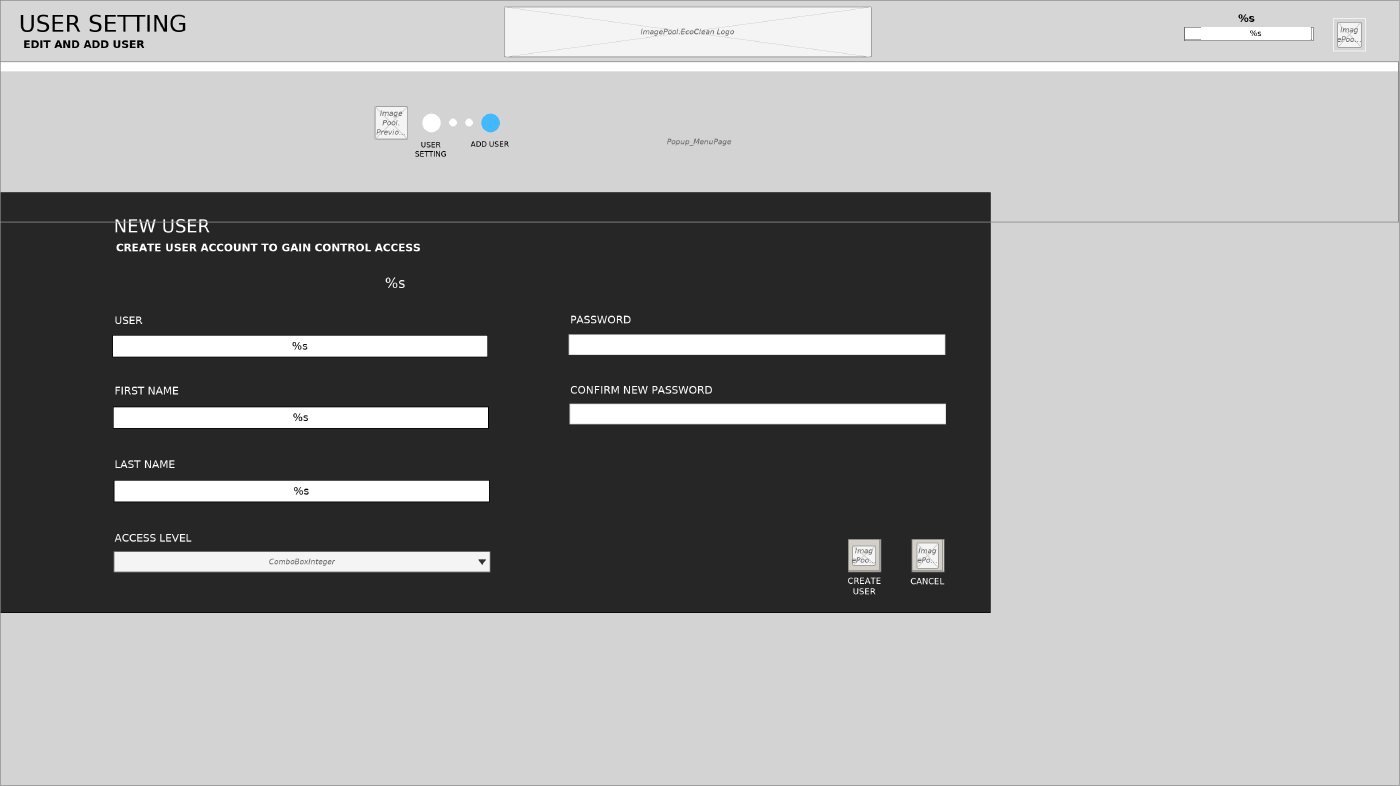
VISUALIZATION AddNewUser_Page  // 1920x1079
    Rectangle (0,98 1920x981)
    Rectangle (0,63 1920x26)
        p3528305787: HMI_Ctrl.ANIMATION3
    Rectangle (0,0 1919x85)
    Label (23,6 310x53), "USER SETTING"
    Label (29,49 320x24), "EDIT AND ADD USER"
    Group (1828,25 45x45)
        OnMouseClick: toggle HMI_Ctrl.MenuButton
        RoundedRectangle (0,0 45x45), colour toggle: HMI_Ctrl.MenuButton
        Image (6,5 33x35), image: ImagePool.Menu Button
    Image (691,9 504x69), image: ImagePool.EcoClean Logo
    Group (1621,14 180x42)
        Rectangle (0,0 177x22), "%s", text variable: DSLocalSystemTimeML.sCurrentDT24Hr_General
        Button (3,23 177x19), image: VisuSymbols.Symbols.AddUser
        Rectangle (26,23 150x18), "%s", text variable: fbHmiTF1800_UserlevelManagement.dsHmiUserStatus_Active.sLoginName
    Rectangle (0,264 1358x577)
    Label (153,284 221x53), "NEW USER"
    Label (156,321 609x38), "CREATE USER ACCOUNT TO GAIN CONTROL ACCESS"
    Label (154,712 216x53), "ACCESS LEVEL"
    ComboBoxInteger (156,757 516x28), variable: sUM_NewUserGroupId, text list: 'TextList_AccessLevel'
    Label (154,611 216x53), "LAST NAME"
    Label (154,409 123x62), "USER"
    Label (154,510 216x53), "FIRST NAME"
    Label (779,408 195x62), "PASSWORD"
    Label (779,509 229x53), "CONFIRM NEW PASSWORD"
    Textfield (781,554 516x28), text variable: sUM_ConfirmPassword
        OnMouseDown: write the text variable via Default, password
    Textfield (780,459 516x28), text variable: sUM_NewPassword
        OnMouseDown: write the text variable via Default, password
    RoundedRectangle (601,151 163x35)
    Ellipse (579,156 25x25)
    Ellipse (660,156 25x25)
    Ellipse (616,163 10x10)
    Ellipse (638,163 10x10)
    Label (559,186 64x39), "USER SETTING"
    Label (640,186 64x24), "ADD USER"
    Image (514,146 45x45), image: ImagePool.Previous Button
        OnMouseClick: change screen: UserSetting_Page
    Group (1155,740 61x86)
        toggle bUM_CreatePB
        Button (8,0 45x45)
        Label (0,44 61x42), "CREATE USER"
        Image (14,9 32x27), image: ImagePool.Add User
    Group (1242,740 60x80)
        toggle bUM_ReturnPB
        Button (8,0 45x45)
        Label (0,36 60x44), "CANCEL"
        Image (15,5 30x35), image: ImagePool.Cancel
    Rectangle (155,558 515x30), "%s", text variable: sUM_NewUserFirstName
        OnMouseDown: write the text variable via Default
    Rectangle (156,659 515x30), "%s", text variable: sUM_NewUserLastName
        OnMouseDown: write the text variable via Default
    Rectangle (154,460 515x30), "%s", text variable: sUM_NewUserLoginName
        OnMouseDown: write the text variable via Default
    Textfield (158,374 768x30), "%s", text variable: sMessage
    Frame (0,84 1918x221), invisible if: HMI_Ctrl.CloseMenuButton
        shows Popup_MenuPage()
END_VISUALIZATION

(* stored: Version 1.1.0.1, ProductVersion 3.1.4024.12
   Visu AddNewUser_Page: Id {87ba9c99-da7e-4f23-8073-d0214724b9b1} *)
